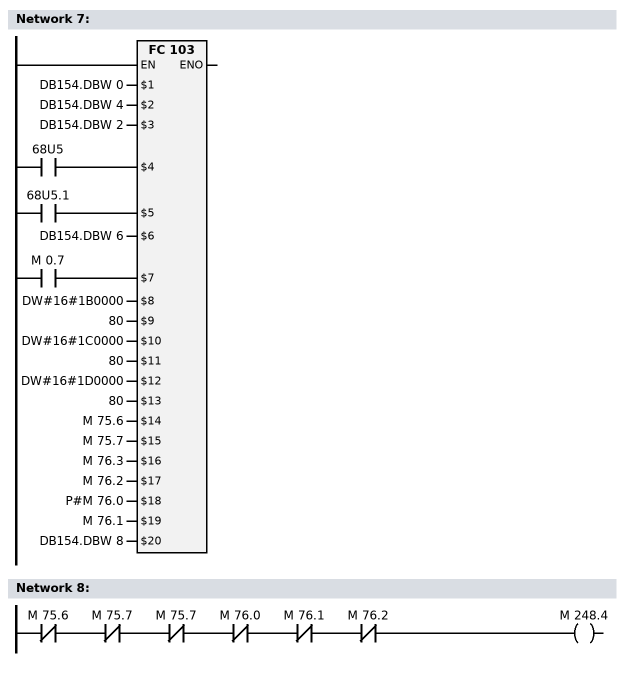
NETWORK
TITLE =
      A     "68U5";
      =     L 52.0;
      BLD   103;
      A     "68U5.1";
      =     L 52.1;
      BLD   103;
      A     M 0.7;
      =     L 52.2;
      BLD   103;
      CALL  FC 103 (
           $1                       := DB154.DBW 0,
           $2                       := DB154.DBW 4,
           $3                       := DB154.DBW 2,
           $4                       := L 52.0,
           $5                       := L 52.1,
           $6                       := DB154.DBW 6,
           $7                       := L 52.2,
           $8                       := DW#16#1B0000,
           $9                       := 80,
           $10                      := DW#16#1C0000,
           $11                      := 80,
           $12                      := DW#16#1D0000,
           $13                      := 80,
           $14                      := M 75.6,
           $15                      := M 75.7,
           $16                      := M 76.3,
           $17                      := M 76.2,
           $18                      := P#M 76.0,
           $19                      := M 76.1,
           $20                      := DB154.DBW 8);
      NOP   0;
NETWORK
TITLE =
      AN    M 75.6;
      AN    M 75.7;
      AN    M 75.7;
      AN    M 76.0;
      AN    M 76.1;
      AN    M 76.2;
      =     M 248.4;
END_FUNCTION

FUNCTION FC 280 : VOID
VERSION : 0.1
BEGIN
// (block stored without names or comments; labels and parameter names are numbered)
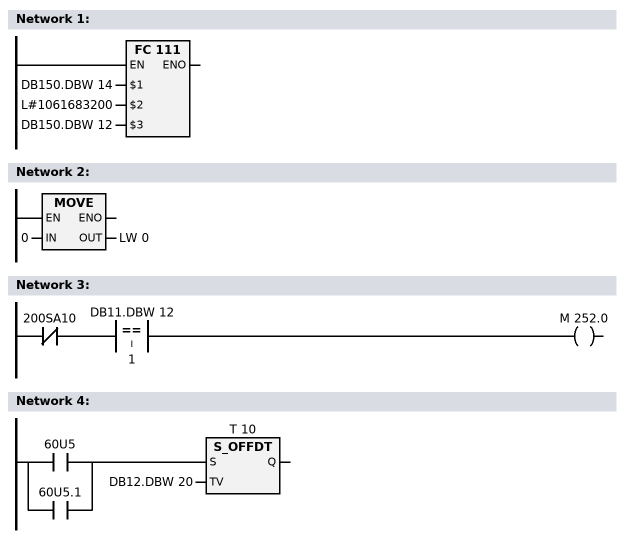
NETWORK
TITLE =
      CALL  FC 111 (
           $1                       := DB150.DBW 14,
           $2                       := L#1061683200,
           $3                       := DB150.DBW 12);
NETWORK
TITLE =
      L     0;
      T     LW 0;
      NOP   0;
NETWORK
TITLE =
      AN    "200SA10";
      A(;
      L     DB11.DBW 12;
      L     1;
      ==I;
      );
      =     M 252.0;
NETWORK
TITLE =
      A(;
      O     "60U5";
      O     "60U5.1";
      );
      L     DB12.DBW 20;
      SF    T 10;
      NOP   0;
      NOP   0;
      NOP   0;
      NOP   0;
NETWORK
TITLE =
      A     M 252.0;
      AN    T 10;
      A     "415SQ7";
      =     L 2.0;
      A     L 2.0;
      BLD   102;
      =     L 0.7;
      A(;
      A     L 2.0;
      JNB   M001;
      L     LW 0;
      T     PQW 260;
      SET;
      SAVE;
      CLR;
M001: A     BR;
      );
      JNB   M002;
      L     DB150.DBW 12;
      T     PQW 262;
      SET;
      SAVE;
      CLR;
M002: A     BR;
      =     L 2.1;
      A     L 2.1;
      BLD   102;
      R     L 0.7;
      A     L 2.1;
      JNB   M003;
      L     LW 0;
      T     PQW 260;
M003: NOP   0;
END_FUNCTION

FUNCTION FC 281 : VOID
VERSION : 0.1
BEGIN
// (block stored without names or comments; labels and parameter names are numbered)
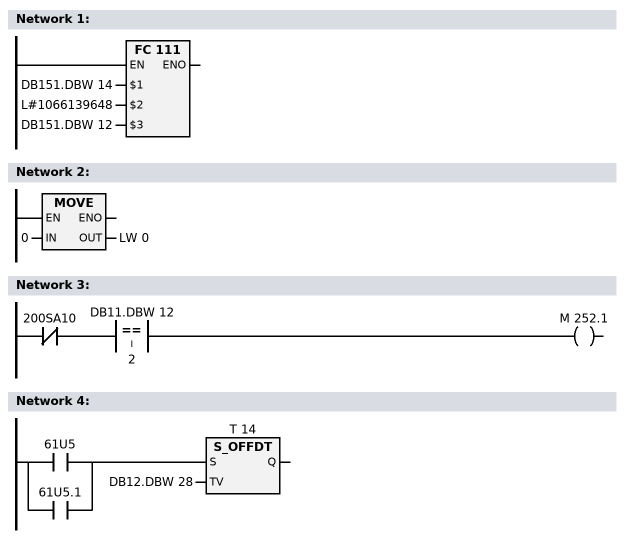
NETWORK
TITLE =
      CALL  FC 111 (
           $1                       := DB151.DBW 14,
           $2                       := L#1066139648,
           $3                       := DB151.DBW 12);
NETWORK
TITLE =
      L     0;
      T     LW 0;
      NOP   0;
NETWORK
TITLE =
      AN    "200SA10";
      A(;
      L     DB11.DBW 12;
      L     2;
      ==I;
      );
      =     M 252.1;
NETWORK
TITLE =
      A(;
      O     "61U5";
      O     "61U5.1";
      );
      L     DB12.DBW 28;
      SF    T 14;
      NOP   0;
      NOP   0;
      NOP   0;
      NOP   0;
NETWORK
TITLE =
      A     M 252.1;
      AN    T 14;
      A     "415SQ6";
      =     L 2.0;
      A     L 2.0;
      BLD   102;
      =     L 0.7;
      A(;
      A     L 2.0;
      JNB   M001;
      L     LW 0;
      T     PQW 256;
      SET;
      SAVE;
      CLR;
M001: A     BR;
      );
      JNB   M002;
      L     DB151.DBW 12;
      T     PQW 258;
      SET;
      SAVE;
      CLR;
M002: A     BR;
      =     L 2.1;
      A     L 2.1;
      BLD   102;
      R     L 0.7;
      A     L 2.1;
      JNB   M003;
      L     LW 0;
      T     PQW 256;
M003: NOP   0;
END_FUNCTION

FUNCTION FC 282 : VOID
VERSION : 0.1
BEGIN
// (block stored without names or comments; labels and parameter names are numbered)
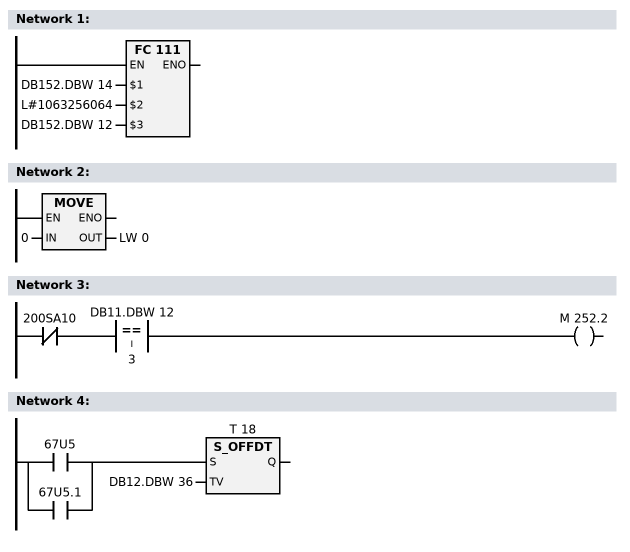
NETWORK
TITLE =
      CALL  FC 111 (
           $1                       := DB152.DBW 14,
           $2                       := L#1063256064,
           $3                       := DB152.DBW 12);
NETWORK
TITLE =
      L     0;
      T     LW 0;
      NOP   0;
NETWORK
TITLE =
      AN    "200SA10";
      A(;
      L     DB11.DBW 12;
      L     3;
      ==I;
      );
      =     M 252.2;
NETWORK
TITLE =
      A(;
      O     "67U5";
      O     "67U5.1";
      );
      L     DB12.DBW 36;
      SF    T 18;
      NOP   0;
      NOP   0;
      NOP   0;
      NOP   0;
NETWORK
TITLE =
      A     M 252.2;
      AN    T 18;
      A     "416SQ3";
      =     L 2.0;
      A     L 2.0;
      BLD   102;
      =     L 0.7;
      A(;
      A     L 2.0;
      JNB   M001;
      L     LW 0;
      T     PQW 272;
      SET;
      SAVE;
      CLR;
M001: A     BR;
      );
      JNB   M002;
      L     DB152.DBW 12;
      T     PQW 274;
      SET;
      SAVE;
      CLR;
M002: A     BR;
      =     L 2.1;
      A     L 2.1;
      BLD   102;
      R     L 0.7;
      A     L 2.1;
      JNB   M003;
      L     LW 0;
      T     PQW 272;
M003: NOP   0;
END_FUNCTION

FUNCTION FC 283 : VOID
VERSION : 0.1
BEGIN
// (block stored without names or comments; labels and parameter names are numbered)
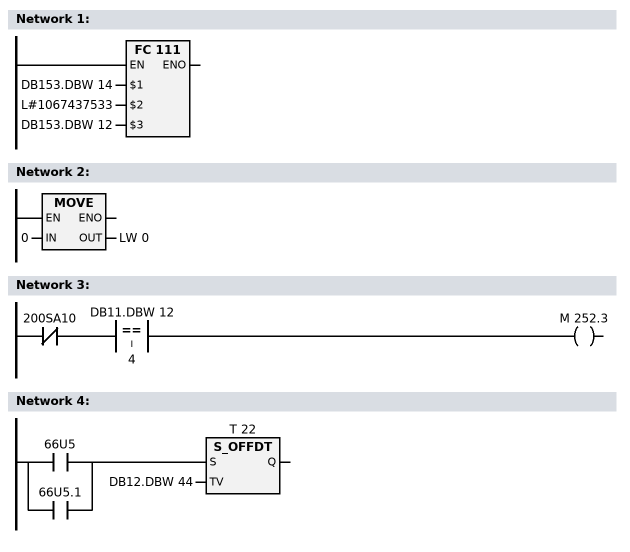
NETWORK
TITLE =
      CALL  FC 111 (
           $1                       := DB153.DBW 14,
           $2                       := L#1067437533,
           $3                       := DB153.DBW 12);
NETWORK
TITLE =
      L     0;
      T     LW 0;
      NOP   0;
NETWORK
TITLE =
      AN    "200SA10";
      A(;
      L     DB11.DBW 12;
      L     4;
      ==I;
      );
      =     M 252.3;
NETWORK
TITLE =
      A(;
      O     "66U5";
      O     "66U5.1";
      );
      L     DB12.DBW 44;
      SF    T 22;
      NOP   0;
      NOP   0;
      NOP   0;
      NOP   0;
NETWORK
TITLE =
      A     M 252.3;
      AN    T 22;
      A     "416SQ2";
      =     L 2.0;
      A     L 2.0;
      BLD   102;
      =     L 0.7;
      A(;
      A     L 2.0;
      JNB   M001;
      L     LW 0;
      T     PQW 268;
      SET;
      SAVE;
      CLR;
M001: A     BR;
      );
      JNB   M002;
      L     DB153.DBW 12;
      T     PQW 270;
      SET;
      SAVE;
      CLR;
M002: A     BR;
      =     L 2.1;
      A     L 2.1;
      BLD   102;
      R     L 0.7;
      A     L 2.1;
      JNB   M003;
      L     LW 0;
      T     PQW 268;
M003: NOP   0;
END_FUNCTION

FUNCTION FC 284 : VOID
VERSION : 0.1
BEGIN
// (block stored without names or comments; labels and parameter names are numbered)
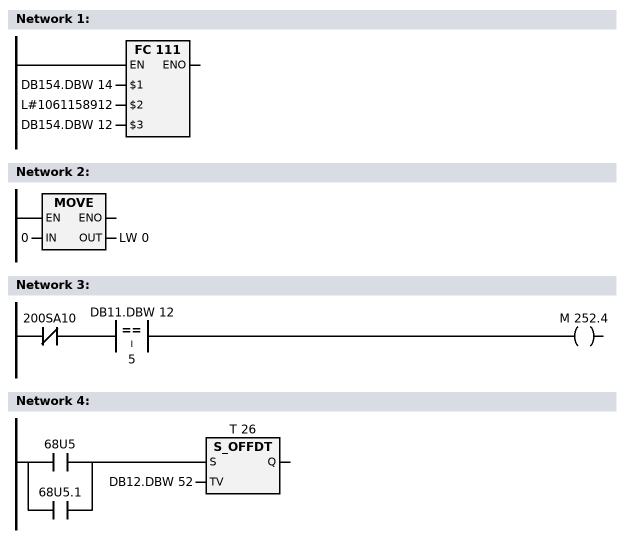
NETWORK
TITLE =
      CALL  FC 111 (
           $1                       := DB154.DBW 14,
           $2                       := L#1061158912,
           $3                       := DB154.DBW 12);
NETWORK
TITLE =
      L     0;
      T     LW 0;
      NOP   0;
NETWORK
TITLE =
      AN    "200SA10";
      A(;
      L     DB11.DBW 12;
      L     5;
      ==I;
      );
      =     M 252.4;
NETWORK
TITLE =
      A(;
      O     "68U5";
      O     "68U5.1";
      );
      L     DB12.DBW 52;
      SF    T 26;
      NOP   0;
      NOP   0;
      NOP   0;
      NOP   0;
NETWORK
TITLE =
      A     M 252.4;
      AN    T 26;
      A     "412SQ5";
      =     L 2.0;
      A     L 2.0;
      BLD   102;
      =     L 0.7;
      A(;
      A     L 2.0;
      JNB   M001;
      L     LW 0;
      T     PQW 264;
      SET;
      SAVE;
      CLR;
M001: A     BR;
      );
      JNB   M002;
      L     DB154.DBW 12;
      T     PQW 266;
      SET;
      SAVE;
      CLR;
M002: A     BR;
      =     L 2.1;
      A     L 2.1;
      BLD   102;
      R     L 0.7;
      A     L 2.1;
      JNB   M003;
      L     LW 0;
      T     PQW 264;
M003: NOP   0;
END_FUNCTION

FUNCTION FC 310 : VOID
VERSION : 0.1
BEGIN
// (block stored without names or comments; labels and parameter names are numbered)
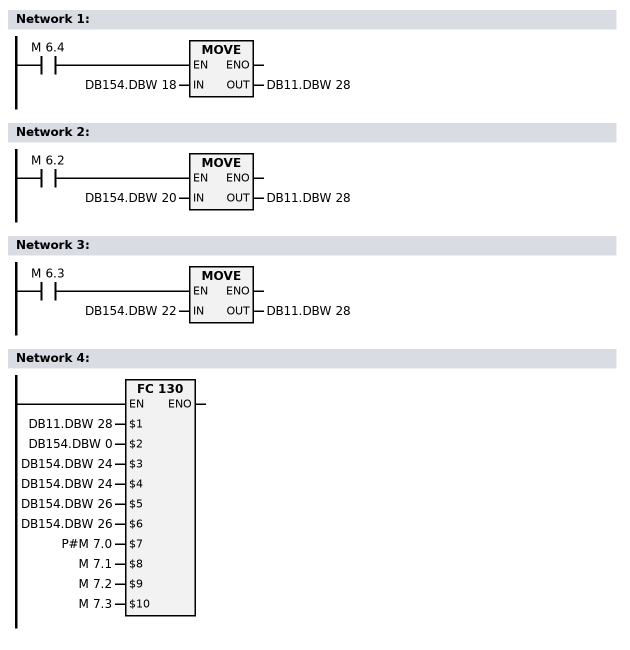
NETWORK
TITLE =
      A     M 6.4;
      JNB   M001;
      L     DB154.DBW 18;
      T     DB11.DBW 28;
M001: NOP   0;
NETWORK
TITLE =
      A     M 6.2;
      JNB   M002;
      L     DB154.DBW 20;
      T     DB11.DBW 28;
M002: NOP   0;
NETWORK
TITLE =
      A     M 6.3;
      JNB   M003;
      L     DB154.DBW 22;
      T     DB11.DBW 28;
M003: NOP   0;
NETWORK
TITLE =
      CALL  FC 130 (
           $1                       := DB11.DBW 28,
           $2                       := DB154.DBW 0,
           $3                       := DB154.DBW 24,
           $4                       := DB154.DBW 24,
           $5                       := DB154.DBW 26,
           $6                       := DB154.DBW 26,
           $7                       := P#M 7.0,
           $8                       := M 7.1,
           $9                       := M 7.2,
           $10                      := M 7.3);
      NOP   0;
END_FUNCTION

FUNCTION FC 311 : VOID
VERSION : 0.1
BEGIN
// (block stored without names or comments; labels and parameter names are numbered)
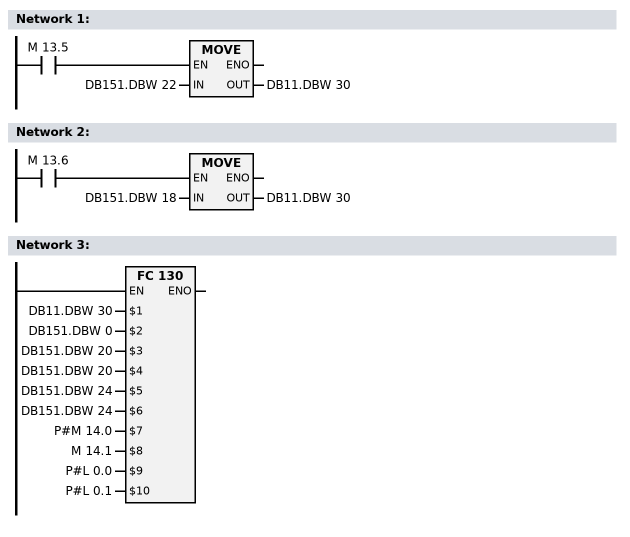
NETWORK
TITLE =
      A     M 13.5;
      JNB   M001;
      L     DB151.DBW 22;
      T     DB11.DBW 30;
M001: NOP   0;
NETWORK
TITLE =
      A     M 13.6;
      JNB   M002;
      L     DB151.DBW 18;
      T     DB11.DBW 30;
M002: NOP   0;
NETWORK
TITLE =
      CALL  FC 130 (
           $1                       := DB11.DBW 30,
           $2                       := DB151.DBW 0,
           $3                       := DB151.DBW 20,
           $4                       := DB151.DBW 20,
           $5                       := DB151.DBW 24,
           $6                       := DB151.DBW 24,
           $7                       := P#M 14.0,
           $8                       := M 14.1,
           $9                       := P#L 0.0,
           $10                      := P#L 0.1);
      NOP   0;
END_FUNCTION

FUNCTION FC 312 : VOID
VERSION : 0.1
BEGIN
// (block stored without names or comments; labels and parameter names are numbered)
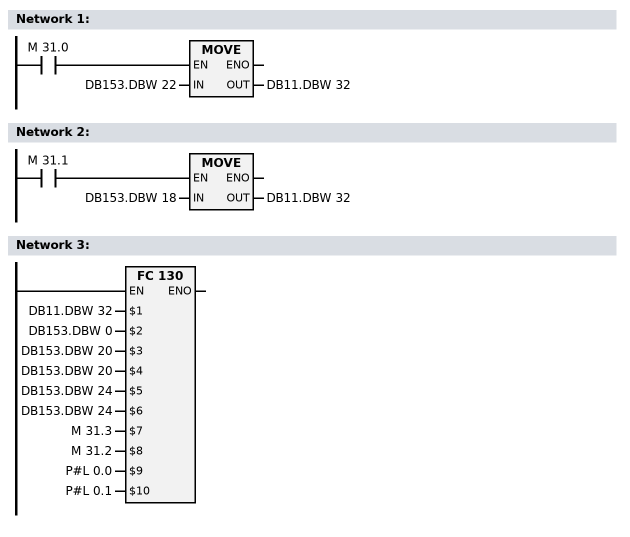
NETWORK
TITLE =
      A     M 31.0;
      JNB   M001;
      L     DB153.DBW 22;
      T     DB11.DBW 32;
M001: NOP   0;
NETWORK
TITLE =
      A     M 31.1;
      JNB   M002;
      L     DB153.DBW 18;
      T     DB11.DBW 32;
M002: NOP   0;
NETWORK
TITLE =
      CALL  FC 130 (
           $1                       := DB11.DBW 32,
           $2                       := DB153.DBW 0,
           $3                       := DB153.DBW 20,
           $4                       := DB153.DBW 20,
           $5                       := DB153.DBW 24,
           $6                       := DB153.DBW 24,
           $7                       := M 31.3,
           $8                       := M 31.2,
           $9                       := P#L 0.0,
           $10                      := P#L 0.1);
      NOP   0;
END_FUNCTION

FUNCTION FC 320 : VOID
VERSION : 0.1
BEGIN
// (block stored without names or comments; labels and parameter names are numbered)
NETWORK
TITLE =
      A(;
      A     M 238.0;
      JNB   M001;
      L     DB11.DBW 70;
      L     150;
      +I;
      T     LW 10;
      AN    OV;
      SAVE;
      CLR;
M001: A     BR;
      );
      A(;
      L     DB150.DBW 0;
      L     LW 10;
      <=I;
      );
      =     L 0.0;
      =     M 12.0;
NETWORK
TITLE =
      A(;
      A     M 238.0;
      JNB   M002;
      L     DB11.DBW 72;
      L     150;
      +I;
      T     LW 12;
      AN    OV;
      SAVE;
      CLR;
M002: A     BR;
      );
      A(;
      L     DB150.DBW 0;
      L     LW 12;
      <=I;
      );
      =     L 0.1;
NETWORK
TITLE =
      A     M 255.0;
      A     "60U5";
      AN    M 200.3;
      AN    M 200.4;
      AN    M 252.0;
      =     L 0.2;
NETWORK
TITLE =
      A     M 255.0;
      A     "60U5";
      A     M 200.3;
      AN    M 200.4;
      AN    M 252.0;
      AN    L 0.2;
      =     L 0.3;
NETWORK
TITLE =
      A     M 255.0;
      A     "60U5.1";
      A(;
      A     M 203.3;
      AN    M 200.2;
      AN    M 200.0;
      AN    L 0.0;
      O;
      A     M 203.1;
      A(;
      AN    M 42.6;
      AN    M 200.5;
      AN    M 200.1;
      AN    L 0.1;
      O;
      A     M 238.0;
      A     M 42.6;
      AN    M 200.5;
      AN    M 200.1;
      );
      );
      AN    M 252.0;
      AN    L 0.5;
      =     L 0.4;
NETWORK
TITLE =
      A     M 255.0;
      A     "60U5.1";
      A(;
      A     M 203.3;
      AN    M 200.0;
      A     L 0.0;
      O;
      A     M 203.1;
      A(;
      AN    M 42.6;
      AN    M 200.1;
      A     L 0.1;
      O;
      A     M 238.0;
      A     M 42.6;
      AN    M 200.1;
      A     M 200.5;
      );
      );
      AN    M 252.0;
      AN    L 0.4;
      =     L 0.5;
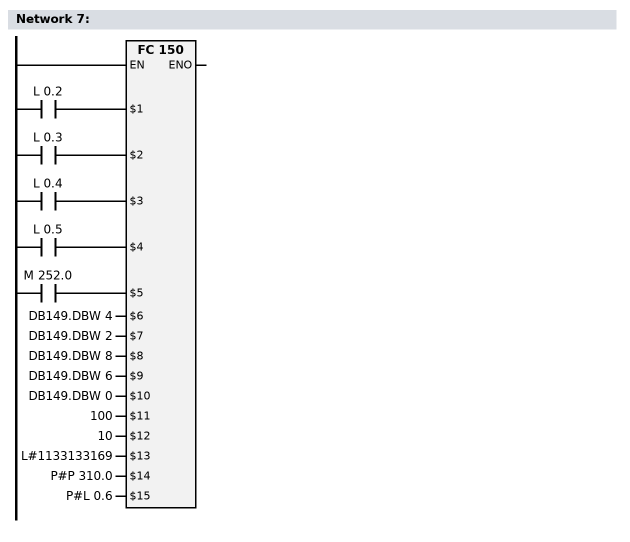
NETWORK
TITLE =
      A     L 0.2;
      =     L 14.0;
      BLD   103;
      A     L 0.3;
      =     L 14.1;
      BLD   103;
      A     L 0.4;
      =     L 14.2;
      BLD   103;
      A     L 0.5;
      =     L 14.3;
      BLD   103;
      A     M 252.0;
      =     L 14.4;
      BLD   103;
      CALL  FC 150 (
           $1                       := L 14.0,
           $2                       := L 14.1,
           $3                       := L 14.2,
           $4                       := L 14.3,
           $5                       := L 14.4,
           $6                       := DB149.DBW 4,
           $7                       := DB149.DBW 2,
           $8                       := DB149.DBW 8,
           $9                       := DB149.DBW 6,
           $10                      := DB149.DBW 0,
           $11                      := 100,
           $12                      := 10,
           $13                      := L#1133133169,
           $14                      := P#P 310.0,
           $15                      := P#L 0.6);
      NOP   0;
END_FUNCTION

FUNCTION FC 321 : VOID
VERSION : 0.1
BEGIN
// (block stored without names or comments; labels and parameter names are numbered)
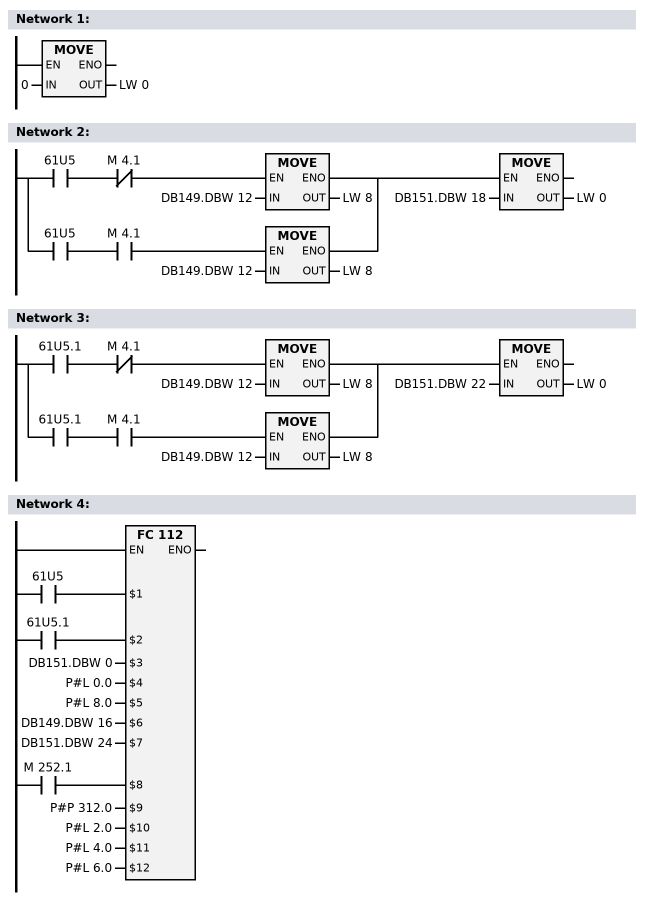
NETWORK
TITLE =
      L     0;
      T     LW 0;
      NOP   0;
NETWORK
TITLE =
      A(;
      O(;
      A     "61U5";
      AN    M 4.1;
      JNB   M001;
      L     DB149.DBW 12;
      T     LW 8;
      SET;
      SAVE;
      CLR;
M001: A     BR;
      );
      O(;
      A     "61U5";
      A     M 4.1;
      JNB   M002;
      L     DB149.DBW 12;
      T     LW 8;
      SET;
      SAVE;
      CLR;
M002: A     BR;
      );
      );
      JNB   M003;
      L     DB151.DBW 18;
      T     LW 0;
M003: NOP   0;
NETWORK
TITLE =
      A(;
      O(;
      A     "61U5.1";
      AN    M 4.1;
      JNB   M004;
      L     DB149.DBW 12;
      T     LW 8;
      SET;
      SAVE;
      CLR;
M004: A     BR;
      );
      O(;
      A     "61U5.1";
      A     M 4.1;
      JNB   M005;
      L     DB149.DBW 12;
      T     LW 8;
      SET;
      SAVE;
      CLR;
M005: A     BR;
      );
      );
      JNB   M006;
      L     DB151.DBW 22;
      T     LW 0;
M006: NOP   0;
NETWORK
TITLE =
      A     "61U5";
      =     L 12.0;
      BLD   103;
      A     "61U5.1";
      =     L 12.1;
      BLD   103;
      A     M 252.1;
      =     L 12.2;
      BLD   103;
      CALL  FC 112 (
           $1                       := L 12.0,
           $2                       := L 12.1,
           $3                       := DB151.DBW 0,
           $4                       := P#L 0.0,
           $5                       := P#L 8.0,
           $6                       := DB149.DBW 16,
           $7                       := DB151.DBW 24,
           $8                       := L 12.2,
           $9                       := P#P 312.0,
           $10                      := P#L 2.0,
           $11                      := P#L 4.0,
           $12                      := P#L 6.0);
      NOP   0;
END_FUNCTION

FUNCTION FC 322 : VOID
VERSION : 0.1
BEGIN
// (block stored without names or comments; labels and parameter names are numbered)
NETWORK
TITLE =
      A     M 255.0;
      A     "67U5";
      AN    M 206.3;
      AN    M 206.4;
      AN    M 252.2;
      =     L 0.2;
NETWORK
TITLE =
      A     M 255.0;
      A     "67U5";
      A     M 206.3;
      AN    M 206.4;
      AN    M 252.2;
      =     L 0.3;
NETWORK
TITLE =
      A     M 255.0;
      A     "67U5.1";
      A(;
      A     M 203.7;
      AN    M 206.5;
      AN    M 206.1;
      AN    "416BF9";
      O;
      A     M 203.5;
      AN    M 206.2;
      AN    M 206.0;
      A     "416SQ8";
      );
      AN    M 252.0;
      =     L 0.4;
NETWORK
TITLE =
      A     M 255.0;
      A     "67U5.1";
      A(;
      A     M 203.7;
      A(;
      O     M 206.5;
      O     "416BF9";
      );
      AN    M 206.1;
      O;
      A     M 203.5;
      A(;
      O     M 206.2;
      ON    "416SQ8";
      );
      AN    M 206.0;
      );
      AN    M 252.0;
      =     L 0.5;
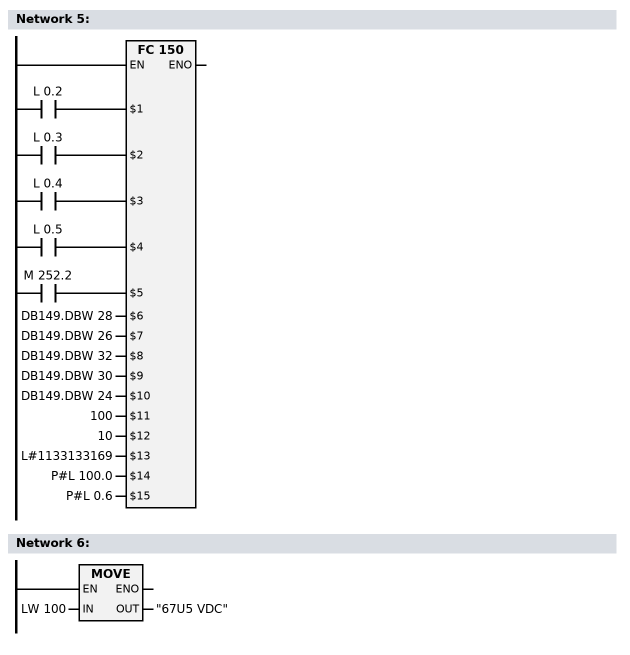
NETWORK
TITLE =
      A     L 0.2;
      =     L 102.0;
      BLD   103;
      A     L 0.3;
      =     L 102.1;
      BLD   103;
      A     L 0.4;
      =     L 102.2;
      BLD   103;
      A     L 0.5;
      =     L 102.3;
      BLD   103;
      A     M 252.2;
      =     L 102.4;
      BLD   103;
      CALL  FC 150 (
           $1                       := L 102.0,
           $2                       := L 102.1,
           $3                       := L 102.2,
           $4                       := L 102.3,
           $5                       := L 102.4,
           $6                       := DB149.DBW 28,
           $7                       := DB149.DBW 26,
           $8                       := DB149.DBW 32,
           $9                       := DB149.DBW 30,
           $10                      := DB149.DBW 24,
           $11                      := 100,
           $12                      := 10,
           $13                      := L#1133133169,
           $14                      := P#L 100.0,
           $15                      := P#L 0.6);
      NOP   0;
NETWORK
TITLE =
      L     LW 100;
      T     "67U5 VDC";
      NOP   0;
END_FUNCTION

FUNCTION FC 323 : VOID
VERSION : 0.1
BEGIN
// (block stored without names or comments; labels and parameter names are numbered)
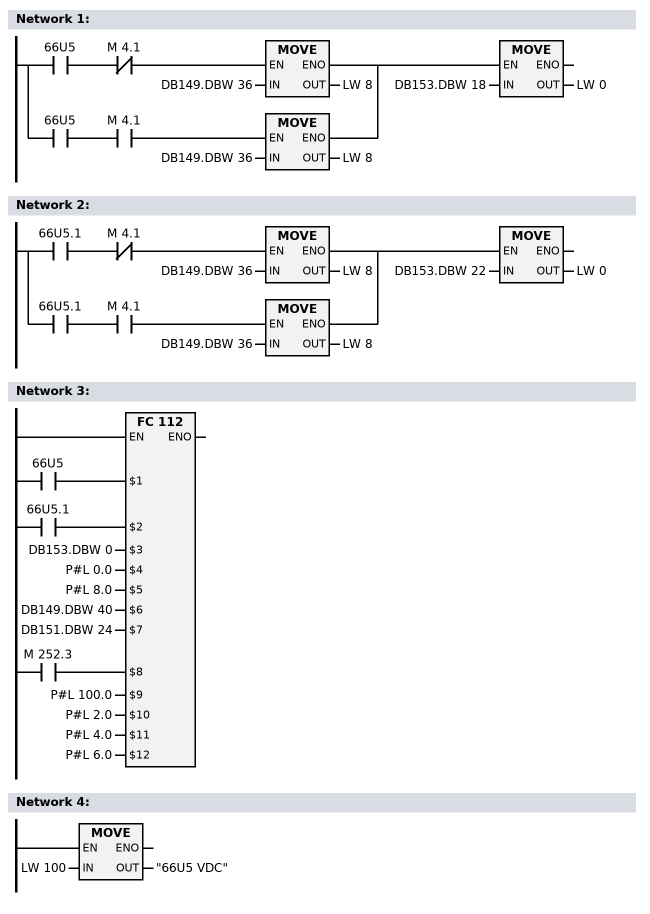
NETWORK
TITLE =
      A(;
      O(;
      A     "66U5";
      AN    M 4.1;
      JNB   M001;
      L     DB149.DBW 36;
      T     LW 8;
      SET;
      SAVE;
      CLR;
M001: A     BR;
      );
      O(;
      A     "66U5";
      A     M 4.1;
      JNB   M002;
      L     DB149.DBW 36;
      T     LW 8;
      SET;
      SAVE;
      CLR;
M002: A     BR;
      );
      );
      JNB   M003;
      L     DB153.DBW 18;
      T     LW 0;
M003: NOP   0;
NETWORK
TITLE =
      A(;
      O(;
      A     "66U5.1";
      AN    M 4.1;
      JNB   M004;
      L     DB149.DBW 36;
      T     LW 8;
      SET;
      SAVE;
      CLR;
M004: A     BR;
      );
      O(;
      A     "66U5.1";
      A     M 4.1;
      JNB   M005;
      L     DB149.DBW 36;
      T     LW 8;
      SET;
      SAVE;
      CLR;
M005: A     BR;
      );
      );
      JNB   M006;
      L     DB153.DBW 22;
      T     LW 0;
M006: NOP   0;
NETWORK
TITLE =
      A     "66U5";
      =     L 102.0;
      BLD   103;
      A     "66U5.1";
      =     L 102.1;
      BLD   103;
      A     M 252.3;
      =     L 102.2;
      BLD   103;
      CALL  FC 112 (
           $1                       := L 102.0,
           $2                       := L 102.1,
           $3                       := DB153.DBW 0,
           $4                       := P#L 0.0,
           $5                       := P#L 8.0,
           $6                       := DB149.DBW 40,
           $7                       := DB151.DBW 24,
           $8                       := L 102.2,
           $9                       := P#L 100.0,
           $10                      := P#L 2.0,
           $11                      := P#L 4.0,
           $12                      := P#L 6.0);
      NOP   0;
NETWORK
TITLE =
      L     LW 100;
      T     "66U5 VDC";
      NOP   0;
END_FUNCTION

DATA_BLOCK DB 5
VERSION : 0.1
BEGIN
// 88 bytes; values not shown
END_DATA_BLOCK

DATA_BLOCK DB 10
VERSION : 0.1
BEGIN
// 40 bytes; values not shown
END_DATA_BLOCK

DATA_BLOCK DB 11
VERSION : 0.1
BEGIN
// 98 bytes; values not shown
END_DATA_BLOCK

DATA_BLOCK DB 12
VERSION : 0.1
BEGIN
// 522 bytes; values not shown
END_DATA_BLOCK

DATA_BLOCK DB 99
VERSION : 0.1
BEGIN
// 210 bytes; values not shown
END_DATA_BLOCK

DATA_BLOCK DB 100
VERSION : 0.1
BEGIN
// 210 bytes; values not shown
END_DATA_BLOCK

DATA_BLOCK DB 101
VERSION : 0.1
BEGIN
// 210 bytes; values not shown
END_DATA_BLOCK

DATA_BLOCK DB 102
VERSION : 0.1
BEGIN
// 210 bytes; values not shown
END_DATA_BLOCK

DATA_BLOCK DB 103
VERSION : 0.1
BEGIN
// 210 bytes; values not shown
END_DATA_BLOCK

DATA_BLOCK DB 149
VERSION : 0.1
BEGIN
// 60 bytes; values not shown
END_DATA_BLOCK

DATA_BLOCK DB 150
VERSION : 0.1
BEGIN
// 40 bytes; values not shown
END_DATA_BLOCK

DATA_BLOCK DB 151
VERSION : 0.1
BEGIN
// 40 bytes; values not shown
END_DATA_BLOCK

DATA_BLOCK DB 152
VERSION : 0.1
BEGIN
// 40 bytes; values not shown
END_DATA_BLOCK

DATA_BLOCK DB 153
VERSION : 0.1
BEGIN
// 40 bytes; values not shown
END_DATA_BLOCK

DATA_BLOCK DB 154
VERSION : 0.1
BEGIN
// 40 bytes; values not shown
END_DATA_BLOCK

ORGANIZATION_BLOCK OB 1
VERSION : 0.1
BEGIN
// (block stored without names or comments; labels and parameter names are numbered)
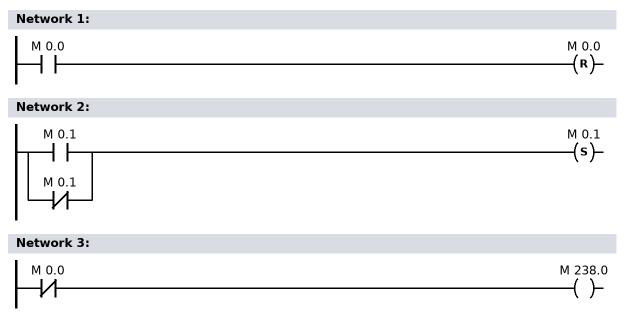
NETWORK
TITLE =
      A     M 0.0;
      R     M 0.0;
NETWORK
TITLE =
      O     M 0.1;
      ON    M 0.1;
      S     M 0.1;
NETWORK
TITLE =
      AN    M 0.0;
      =     M 238.0;
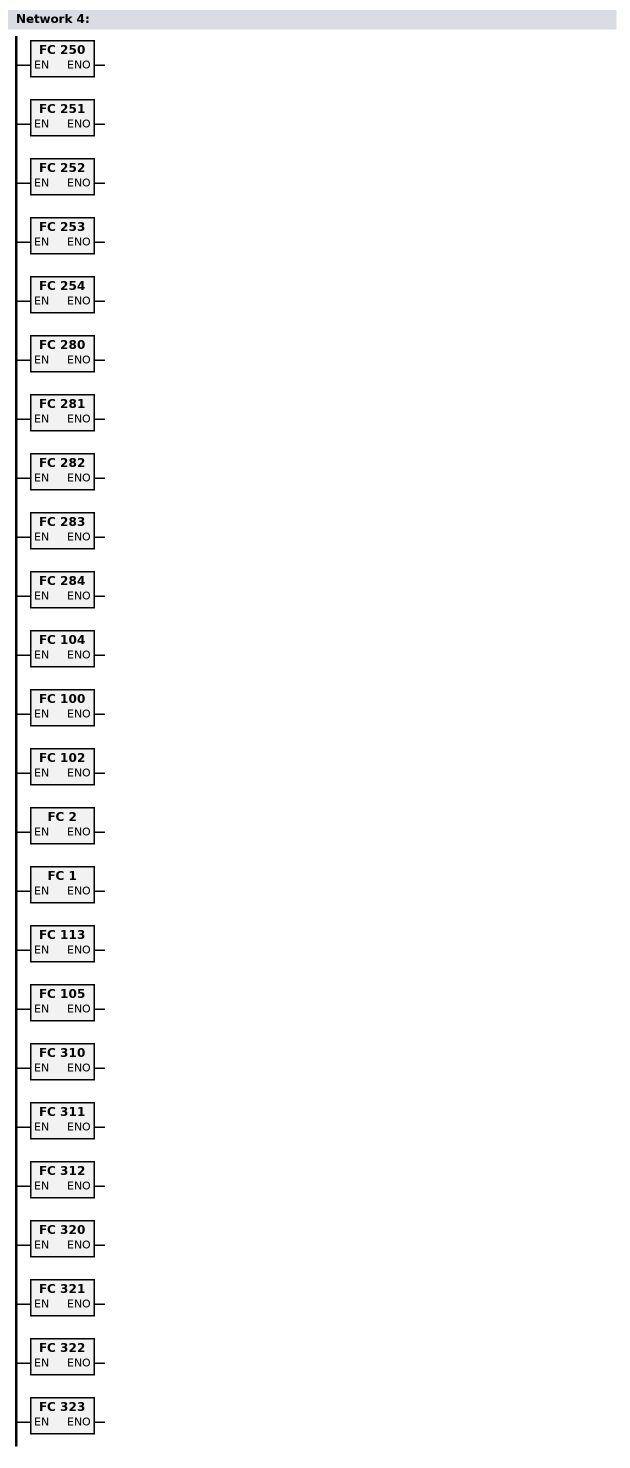
NETWORK
TITLE =
      CALL  FC 250;
      CALL  FC 251;
      CALL  FC 252;
      CALL  FC 253;
      CALL  FC 254;
      CALL  FC 280;
      CALL  FC 281;
      CALL  FC 282;
      CALL  FC 283;
      CALL  FC 284;
      CALL  FC 104;
      CALL  FC 100;
      CALL  FC 102;
      CALL  FC 2;
      CALL  FC 1;
      CALL  FC 113;
      CALL  FC 105;
      CALL  FC 310;
      CALL  FC 311;
      CALL  FC 312;
      CALL  FC 320;
      CALL  FC 321;
      CALL  FC 322;
      CALL  FC 323;
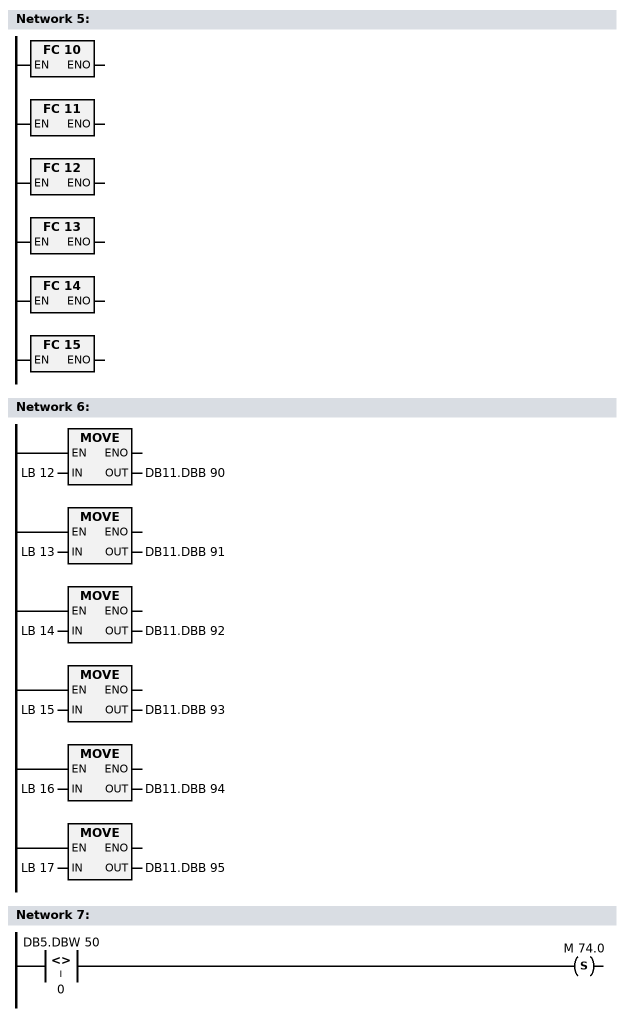
NETWORK
TITLE =
      CALL  FC 10;
      CALL  FC 11;
      CALL  FC 12;
      CALL  FC 13;
      CALL  FC 14;
      CALL  FC 15;
NETWORK
TITLE =
      L     LB 12;
      T     DB11.DBB 90;
      L     LB 13;
      T     DB11.DBB 91;
      L     LB 14;
      T     DB11.DBB 92;
      L     LB 15;
      T     DB11.DBB 93;
      L     LB 16;
      T     DB11.DBB 94;
      L     LB 17;
      T     DB11.DBB 95;
NETWORK
TITLE =
      L     DB5.DBW 50;
      L     0;
      <>I;
      S     M 74.0;
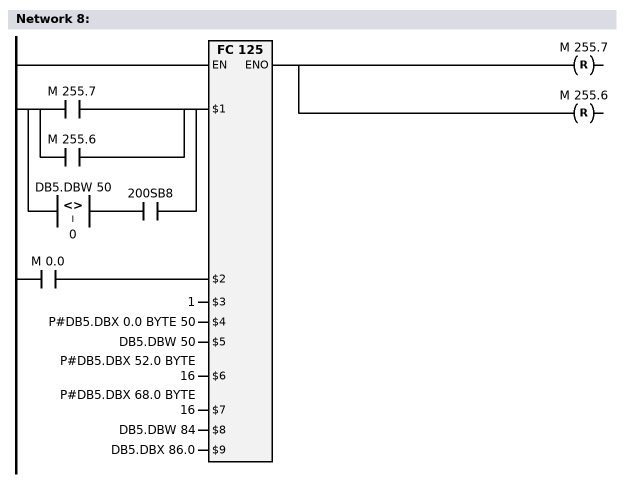
NETWORK
TITLE =
      A(;
      O     M 255.7;
      O     M 255.6;
      O;
      A(;
      L     DB5.DBW 50;
      L     0;
      <>I;
      );
      A     "200SB8";
      );
      =     L 20.0;
      BLD   103;
      A     M 0.0;
      =     L 20.1;
      BLD   103;
      CALL  FC 125 (
           $1                       := L 20.0,
           $2                       := L 20.1,
           $3                       := 1,
           $4                       := P#DB5.DBX 0.0 BYTE 50,
           $5                       := DB5.DBW 50,
           $6                       := P#DB5.DBX 52.0 BYTE 16,
           $7                       := P#DB5.DBX 68.0 BYTE 16,
           $8                       := DB5.DBW 84,
           $9                       := DB5.DBX 86.0);
      A     BR;
      R     M 255.7;
      R     M 255.6;
END_ORGANIZATION_BLOCK

ORGANIZATION_BLOCK OB 82
VERSION : 0.1
BEGIN
// (block stored without names or comments; labels and parameter names are numbered)
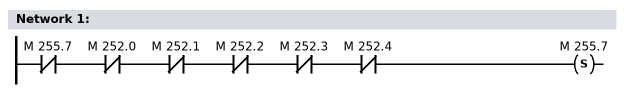
NETWORK
TITLE =
      AN    M 255.7;
      AN    M 252.0;
      AN    M 252.1;
      AN    M 252.2;
      AN    M 252.3;
      AN    M 252.4;
      S     M 255.7;
END_ORGANIZATION_BLOCK

ORGANIZATION_BLOCK OB 86
VERSION : 0.1
BEGIN
// (block stored without names or comments; labels and parameter names are numbered)
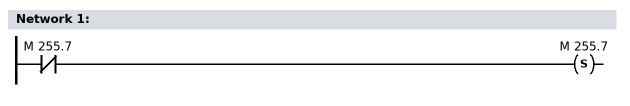
NETWORK
TITLE =
      AN    M 255.7;
      S     M 255.7;
END_ORGANIZATION_BLOCK

ORGANIZATION_BLOCK OB 100
VERSION : 0.0
BEGIN
// (block stored without names or comments; labels and parameter names are numbered)
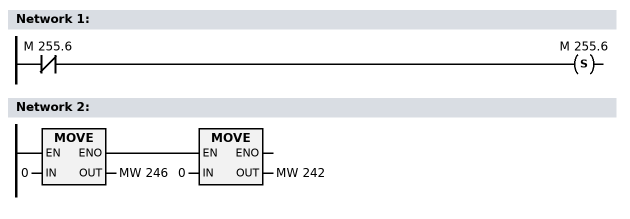
NETWORK
TITLE =
      AN    M 255.6;
      S     M 255.6;
NETWORK
TITLE =
      A(;
      L     0;
      T     MW 246;
      SET;
      SAVE;
      CLR;
      A     BR;
      );
      JNB   M001;
      L     0;
      T     MW 242;
M001: NOP   0;
END_ORGANIZATION_BLOCK

ORGANIZATION_BLOCK OB 121
VERSION : 0.1
BEGIN
// (block stored without names or comments; labels and parameter names are numbered)
NETWORK
TITLE =
END_ORGANIZATION_BLOCK

ORGANIZATION_BLOCK OB 122
VERSION : 0.1
BEGIN
// (block stored without names or comments; labels and parameter names are numbered)
NETWORK
TITLE =
END_ORGANIZATION_BLOCK
